FUNCTION_BLOCK Stack
VAR_INPUT
END_VAR
VAR_OUTPUT
	o_slidingCylinder : MonostableCylinder;
END_VAR
VAR
	//Sensors
	m_Presencesensor : PresenceSensor;
	m_Opticalsensor : OpticalSensor;
	m_Inductivesensor : InductiveSensor;
	m_Weightsensor : WeightSensor;
END_VAR

PROPERTY LightWPOnTray : BOOL
GET
LightWPOnTray:=m_Opticalsensor.Value;
END_GET
END_PROPERTY

PROPERTY MetalWPOnTray : BOOL
GET
MetalWPOnTray := m_Inductivesensor.Value;
END_GET
END_PROPERTY

PROPERTY WPOnTray : BOOL
 //REFERENCE TO PresenceSensor
GET
WPOnTray:=m_Presencesensor.Value;
END_GET
END_PROPERTY

PROPERTY WPWeight : INT
GET
WPWeight:=m_Weightsensor.Value;
END_GET
END_PROPERTY

END_FUNCTION_BLOCK

(* stored: Version 1.1.0.1, ProductVersion 3.1.4024.9
   POU Stack: Id {1ba1d180-29b9-4e18-8f68-aea496937208}, SpecialFunc None
   Property LightWPOnTray: Id {1148e582-0267-4b41-a393-abcf34cda5c6}
   Get Get: Id {c801094a-3827-441d-bea9-9818937fce9b}
   Property MetalWPOnTray: Id {bae225bd-1f2b-44f8-a54c-dc6c67026140}
   Get Get: Id {881015d3-0c8d-4885-a336-31633d321048}
   Property WPOnTray: Id {84c3a07b-ee51-4f44-9348-c1619ae2e8e7}
   Get Get: Id {94bd6cbf-8fd0-4af9-9af5-b15b81d73c12}
   Property WPWeight: Id {77d9348d-54ec-47d0-acec-31def8ad1be8}
   Get Get: Id {c83f1a12-1820-46cb-9224-c9dfd54c27a6} *)
